GLOBALCONSTANTS PKP_2200_LI_DI (* logiBUS_DI constants *)
  (* Standard: 61499-1; Description: Copyright (c) 2024 HR Agrartechnik GmbH This program and the accompanying materials are made available under the terms of the Eclipse Public License 2.0 which is available at https://www.eclipse.org/legal/epl-2.0/ SPDX-License-Identifier: EPL-2.0 *)
  (* Version 1.0, 2024-01-25, Franz Höpfinger, HR Agrartechnik GmbH *)
  VAR_GLOBAL CONSTANT
    DigitalInput_Key_1 : PKP_2200_LI_DI_S := (Pin := 1);
    DigitalInput_Key_2 : PKP_2200_LI_DI_S := (Pin := 2);
    DigitalInput_Key_3 : PKP_2200_LI_DI_S := (Pin := 3);
    DigitalInput_Key_4 : PKP_2200_LI_DI_S := (Pin := 4);
    Invalid : PKP_2200_LI_DI_S := (Pin := 255);
  END_VAR
END_GLOBALCONSTANTS
